// TIA Portal V20 export
DATA_BLOCK "PM05"   // DB233
// stored: MemoryReserve 100
   VAR
      "ANODE GLASS CLEANING ON" : Bool := FALSE;
      SPARE : Bool := FALSE;
      "ANODE MAIN NG P&P UP" : Bool := FALSE;
      "ANODE MAIN NG P&P DOWN" : Bool := FALSE;
      "ANODE MAIN NG P&P 1st FORWARD" : Bool := FALSE;
      "ANODE MAIN NG P&P 1st BACKWARD" : Bool := FALSE;
      "ANODE MAIN NG P&P 2nd FORWARD" : Bool := FALSE;
      "ANODE MAIN NG P&P 2nd BACKWARD" : Bool := FALSE;
      "ANODE FIX FRONT FORWARD / ANODE FIX REAR FORWARD" : Bool := FALSE;
      "ANODE FIX FRONT BACKWARD / ANODE FIX REAR BACKWARD" : Bool := FALSE;
      "ANODE MAIN P&P#1 Rotary CW" : Bool := FALSE;
      "ANODE MAIN P&P#1 Rotary CCW" : Bool := FALSE;
      "ANODE NG BOX LIFT UP" : Bool := FALSE;
      "ANODE NG BOX LIFT DOWN" : Bool := FALSE;
      "ANODE NG BOX LOCK UP" : Bool := FALSE;
      "ANODE NG BOX LOCK DOWN" : Bool := FALSE;
   END_VAR
BEGIN
END_DATA_BLOCK
